// TIA Portal V16 export
// export: Created 2021-11-12T13:32:41.9009173Z, ExportSetting WithDefaults, DisplayName Totally Integrated Automation Portal, DisplayVersion V16 Update 3, DisplayName TIA Portal Version Control Interface, DisplayVersion V16 Update 2, DisplayName TIA Portal Openness, DisplayVersion V16 Update 3, DisplayName SINAMICS Startdrive Advanced, DisplayVersion V16 Update 5, DisplayName SINAMICS Startdrive G130, G150, S120, S150, SINAMICS MV, S210, DisplayVersion V16 Update 5, DisplayName SINAMICS Startdrive G110M, G120, G120C, G120D, G120P, G115D, DisplayVersion V16 Update 5, DisplayName STEP 7 Professional, DisplayVersion V16 Update 3, DisplayName STEP 7 Safety, DisplayVersion V16, DisplayName WinCC UA Professional, DisplayVersion V16 Update 3
DATA_BLOCK "HMI_CMD_200+UH11"   // DB55
{ S7_Optimized_Access := 'TRUE' }
VERSION : 0.1
// stored: AutoNumber true, DBAccessibleFromOPCUA true, IsOnlyStoredInLoadMemory false, IsRetainMemResEnabled false, IsWriteProtectedInAS false, MemoryReserve 100
   VAR
      xxxxx___BinarySensors___xxxxx : Byte;
      xxxxx___BinaryOthers___xxxxx : Byte;
      SF02_14 { S7_SetPoint := 'True'} : "UDT_CH_DI_Command";   // Start automat
      SF03_14 { S7_SetPoint := 'True'} : "UDT_CH_DI_Command";   // Nulování poruchy
      SF04_14 { S7_SetPoint := 'True'} : "UDT_CH_DI_Command";   // Reset bezpečnostního okruhu
      SF05_22 { S7_SetPoint := 'True'} : "UDT_CH_DI_Command";   // Blokování pásu v peci 3
      SF06_22 { S7_SetPoint := 'True'} : "UDT_CH_DI_Command";   // Blokování pásu v peci 1
      SF07_22 { S7_SetPoint := 'True'} : "UDT_CH_DI_Command";   // Blokování pásu v peci 2
      "I450.6" { S7_SetPoint := 'True'} : "UDT_CH_DI_Command";   // Rezerva
      "I450.7" { S7_SetPoint := 'True'} : "UDT_CH_DI_Command";   // Rezerva Okamžitý stop Robot 2R3
      "I451.0" { S7_SetPoint := 'True'} : "UDT_CH_DI_Command";   // Rezerva Okamžitý stop Robot 2R4
      "I451.1" { S7_SetPoint := 'True'} : "UDT_CH_DI_Command";   // Rezerva Okamžitý stop Robot 2R5
      "I451.2" { S7_SetPoint := 'True'} : "UDT_CH_DI_Command";   // Rezerva Okamžitý stop Robot 2R6
      "200UF01-SF02_14" { S7_SetPoint := 'True'} : "UDT_CH_DI_Command";   // Bedna Žádost o výměnu
      "200UF01-SF03_14" { S7_SetPoint := 'True'} : "UDT_CH_DI_Command";   // Bedna Vyměněna
      "I451.5" { S7_SetPoint := 'True'} : "UDT_CH_DI_Command";   // Rezerva Vzorek na test
      "I451.6" { S7_SetPoint := 'True'} : "UDT_CH_DI_Command";   // Rezerva Materiál vložit
      "I451.7" { S7_SetPoint := 'True'} : "UDT_CH_DI_Command";   // Rezerva
      xxxxx___AnalogueSensors___xxxxx : Byte;
      xxxxx___Drives___xxxxx : Byte;
      xxxxx___Other___xxxxx : Byte;
      xxxxx___Alarms___xxxxx : Byte;
      ES : "UDT_DI_Mon_Command";   // E-stop
      KF31 : "UDT_DI_Mon_Command";   // module 200UH11- KF31
   END_VAR
BEGIN
END_DATA_BLOCK
